FUNCTION F_HelloWorld
VAR_INPUT
END_VAR
VAR
	run: BOOL;
END_VAR

IF NOT run THEN
		ADSLOGSTR(msgCtrlMask := ADSLOG_MSGTYPE_ERROR OR ADSLOG_MSGTYPE_LOG,
			msgFmtStr:= 'Hello world!!',
			strArg:='');
			
		run := TRUE;
END_IF

END_FUNCTION

(* stored: Version 1.1.0.1, ProductVersion 3.1.4024.16
   POU F_HelloWorld: Id {1b71dbe9-7d4c-445d-a8d7-fc2fe923832d}, SpecialFunc None *)
